FUNCTION_BLOCK MOVING_AVERAGE
  {SET_ATTRIBUTE(OpcUa, SERVICE)}
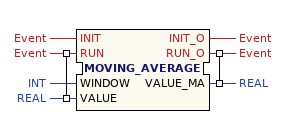
  EVENT_INPUT
    INIT;
    RUN WITH VALUE; {SET_ATTRIBUTE(OpcUa, Method)}
  END_EVENT
  EVENT_OUTPUT
    INIT_O;
    RUN_O WITH VALUE_MA;
  END_EVENT
  VAR_INPUT
    WINDOW : INT; {SET_ATTRIBUTE(OpcUa, Constant.RUN)}
    VALUE : REAL; {SET_ATTRIBUTE(OpcUa, Variable.RUN)}
  END_VAR
  VAR_OUTPUT
    VALUE_MA : REAL; {SET_ATTRIBUTE(OpcUa, Variable.RUN)}
  END_VAR
END_FUNCTION_BLOCK
